FUNCTION_BLOCK FB_XpMoveZ
VAR_IN_OUT
	XpMover							: MC_PlanarMover;
END_VAR
VAR_INPUT
	execute							: BOOL;
	position						: LREAL := 2;
	velocity						: LREAL := 100;
	acceleration					: LREAL := 2000;
	jerk							: LREAL := 20000;
END_VAR
VAR_OUTPUT
	done							: BOOL;
	busy							: BOOL;
	error							: BOOL;
	aborted							: BOOL;
END_VAR
VAR
	_XpFeedback						: ARRAY [0.._MAX_XPLANAR_FEEDBACK] OF MC_PlanarFeedback;
	_XpCondition		 			: DynamicConstraint_Coordinates;
END_VAR
VAR
	_sequence						: UINT;
	_i								: UINT;
	_countError						: UINT;
	_position						: LREAL;
	_velocity						: LREAL;
	_acceleration					: LREAL;
	_jerk							: LREAL;
END_VAR
VAR CONSTANT
	_MAX_XPLANAR_FEEDBACK			: UINT := 1;
	_MAX_COUNT_ERROR				: UINT := 5;
	
	_INIT							: UINT := 0000;
	_READY							: UINT := 0001;
	_MOVE_Z							: UINT := 0011;
	_CHECK_MOVE_Z					: UINT := 0012;
	_DONE							: UINT := 1000;
	_ERROR							: UINT := 2000;
	_ABORTED						: UINT := 3000;
END_VAR

updateXPlanarFB();
CASE _sequence OF
	_INIT:
		_XpCondition.AddLimit(
			Coordinate:= Coord_Mcs_Z, 
			V:= velocity, 
			A:= acceleration, 
			D:= acceleration, 
			J:= jerk);
		_sequence := _READY;
	
	_READY:
		IF execute THEN
			busy := TRUE;
			_sequence := _MOVE_Z;
			setInputVariables();
		END_IF
		
	_MOVE_Z:
		_XpCondition.SetLimit(
			Coordinate:= Coord_Mcs_Z, 
			V:= _velocity, 
			A:= _acceleration, 
			D:= _acceleration, 
			J:= _jerk);
		XpMover.MoveZ(commandFeedback:= _XpFeedback[0], 
			targetPosition:= _position, 
			constraint:= _XpCondition);
		_sequence := _CHECK_MOVE_Z;
		
	_CHECK_MOVE_Z:
		IF _XpFeedback[0].Done THEN
			_countError := 0;
			_sequence := _DONE;
		ELSIF _XpFeedback[0].Error THEN
			_countError := _countError + 1;
			_sequence := _MOVE_Z;
		END_IF
		IF _countError > _MAX_COUNT_ERROR THEN
			_countError := 0;
			_sequence := _ERROR;
		END_IF
		
	_DONE:
		done := TRUE;
		busy := FALSE;
		IF NOT execute THEN
			done := FALSE;
			_sequence := _READY;
		END_IF
	
	_ERROR:
		error := TRUE;
		busy := FALSE;
		IF NOT execute THEN
			error := FALSE;
			_sequence := _READY;
		END_IF
		
	_ABORTED:
		aborted := TRUE;
		busy := FALSE;
		IF NOT execute THEN
			aborted := FALSE;
			_sequence := _READY;
		END_IF
END_CASE

ACTION setInputVariables:
_position := position;
_velocity := velocity;
_acceleration := acceleration;
_jerk := jerk;
END_ACTION

ACTION updateXPlanarFB:
FOR _i:=0 TO _MAX_XPLANAR_FEEDBACK DO
	_XpFeedback[_i].Update();
END_FOR
END_ACTION

END_FUNCTION_BLOCK

(* stored: Version 1.1.0.1
   POU FB_XpMoveZ: Id {74b4c25c-281d-451a-af40-76cf9201cf55}, SpecialFunc None
   Action setInputVariables: Id {66476d73-400d-4622-850d-f10cd64316a1}
   Action updateXPlanarFB: Id {97e29cb9-0b01-47f0-b36b-b4a15a15ca05} *)
